TYPE ST_DwellTime :
STRUCT
	DwellTime	: TIME;
	BufferMode	: MC_BUFFER_MODE := mcBuffered;
	InvokeId	: UDINT;
END_STRUCT
END_TYPE

(* stored: Version 1.1.0.1, ProductVersion 3.1.4024.12
   DUT ST_DwellTime: Id {43cb479e-556c-4d2c-bc55-3b35ecbb9fe1} *)
